// TIA Portal V20 export
TYPE "UDT_BinMon08"
TITLE = MTPDataObjectSUCLibrary/DataAssembly/Indicator/Element/BinMon08
   STRUCT
      V1State0 { ExternalAccessible := 'False'; ExternalVisible := 'False'; ExternalWritable := 'False'} : String[16] := '';   // Text replacement for V1 false
      V1State1 { ExternalAccessible := 'False'; ExternalVisible := 'False'; ExternalWritable := 'False'} : String[16] := '';   // Text replacement for V1 true
      V2State0 { ExternalAccessible := 'False'; ExternalVisible := 'False'; ExternalWritable := 'False'} : String[16] := '';   // Text replacement for V2 false
      V2State1 { ExternalAccessible := 'False'; ExternalVisible := 'False'; ExternalWritable := 'False'} : String[16] := '';   // Text replacement for V2 true
      V3State0 { ExternalAccessible := 'False'; ExternalVisible := 'False'; ExternalWritable := 'False'} : String[16] := '';   // Text replacement for V3 false
      V3State1 { ExternalAccessible := 'False'; ExternalVisible := 'False'; ExternalWritable := 'False'} : String[16] := '';   // Text replacement for V3 true
      V4State0 { ExternalAccessible := 'False'; ExternalVisible := 'False'; ExternalWritable := 'False'} : String[16] := '';   // Text replacement for V4 false
      V4State1 { ExternalAccessible := 'False'; ExternalVisible := 'False'; ExternalWritable := 'False'} : String[16] := '';   // Text replacement for V4 true
      V5State0 { ExternalAccessible := 'False'; ExternalVisible := 'False'; ExternalWritable := 'False'} : String[16] := '';   // Text replacement for V5 false
      V5State1 { ExternalAccessible := 'False'; ExternalVisible := 'False'; ExternalWritable := 'False'} : String[16] := '';   // Text replacement for V5 true
      V6State0 { ExternalAccessible := 'False'; ExternalVisible := 'False'; ExternalWritable := 'False'} : String[16] := '';   // Text replacement for V6 false
      V6State1 { ExternalAccessible := 'False'; ExternalVisible := 'False'; ExternalWritable := 'False'} : String[16] := '';   // Text replacement for V6 true
      V7State0 { ExternalAccessible := 'False'; ExternalVisible := 'False'; ExternalWritable := 'False'} : String[16] := '';   // Text replacement for V7 false
      V7State1 { ExternalAccessible := 'False'; ExternalVisible := 'False'; ExternalWritable := 'False'} : String[16] := '';   // Text replacement for V7 true
      V8State0 { ExternalAccessible := 'False'; ExternalVisible := 'False'; ExternalWritable := 'False'} : String[16] := '';   // Text replacement for V8 false
      V8State1 { ExternalAccessible := 'False'; ExternalVisible := 'False'; ExternalWritable := 'False'} : String[16] := '';   // Text replacement for V8 true
      OSLevel : Byte := 16#00;   // OSLevel variable
      WQC { ExternalWritable := 'False'} : Byte := 16#FF;   // Worst Quality Code variable
      V1 { ExternalWritable := 'False'} : Bool := FALSE;   // Value 1
      V2 { ExternalWritable := 'False'} : Bool := FALSE;   // Value 2
      V3 { ExternalWritable := 'False'} : Bool := FALSE;   // Value 3
      V4 { ExternalWritable := 'False'} : Bool := FALSE;   // Value 4
      V5 { ExternalWritable := 'False'} : Bool := FALSE;   // Value 5
      V6 { ExternalWritable := 'False'} : Bool := FALSE;   // Value 6
      V7 { ExternalWritable := 'False'} : Bool := FALSE;   // Value 7
      V8 { ExternalWritable := 'False'} : Bool := FALSE;   // Value 8
      V1FlutEn { ExternalWritable := 'False'} : Bool;   // Enable Fluttering Recognition1: enabled; 0: disabled
      V1FlutTi : Real;   // Period of an active signal before it will be recognized as flutter-free, in s
      V2FlutEn { ExternalWritable := 'False'} : Bool;   // Enable Fluttering Recognition1: enabled; 0: disabled
      V2FlutTi : Real;   // Period of an active signal before it will be recognized as flutter-free, in s
      V3FlutEn { ExternalWritable := 'False'} : Bool;   // Enable Fluttering Recognition1: enabled; 0: disabled
      V3FlutTi : Real;   // Period of an active signal before it will be recognized as flutter-free, in s
      V4FlutEn { ExternalWritable := 'False'} : Bool;   // Enable Fluttering Recognition1: enabled; 0: disabled
      V4FlutTi : Real;   // Period of an active signal before it will be recognized as flutter-free, in s
      V5FlutEn { ExternalWritable := 'False'} : Bool;   // Enable Fluttering Recognition1: enabled; 0: disabled
      V5FlutTi : Real;   // Period of an active signal before it will be recognized as flutter-free, in s
      V6FlutEn { ExternalWritable := 'False'} : Bool;   // Enable Fluttering Recognition1: enabled; 0: disabled
      V6FlutTi : Real;   // Period of an active signal before it will be recognized as flutter-free, in s
      V7FlutEn { ExternalWritable := 'False'} : Bool;   // Enable Fluttering Recognition1: enabled; 0: disabled
      V7FlutTi : Real;   // Period of an active signal before it will be recognized as flutter-free, in s
      V8FlutEn { ExternalWritable := 'False'} : Bool;   // Enable Fluttering Recognition1: enabled; 0: disabled
      V8FlutTi : Real;   // Period of an active signal before it will be recognized as flutter-free, in s
   END_STRUCT;
END_TYPE
